{attribute 'GeneratedUsingTerminal: EPP3632-0001-0016'}
{attribute addProperty BoxType "EPP3632-0001-0016"}
{attribute addProperty Id "STATUSAT %I*STATUS_B07533568"}
{attribute addProperty CRC "1971471493"}
{attribute addProperty Size "8"}
TYPE Ch2_Status_75824485 :
STRUCT
	{attribute addProperty Name "STATUS"}
	STATUS AT %I* : STATUS_B0753356;
END_STRUCT
END_TYPE

(* stored: Version 1.2.0.0, ProductVersion 3.1.4024.9
   DUT Ch2_Status_75824485: Id {6648adf7-ec32-4ce1-bbe3-f5385a220d5f} *)
